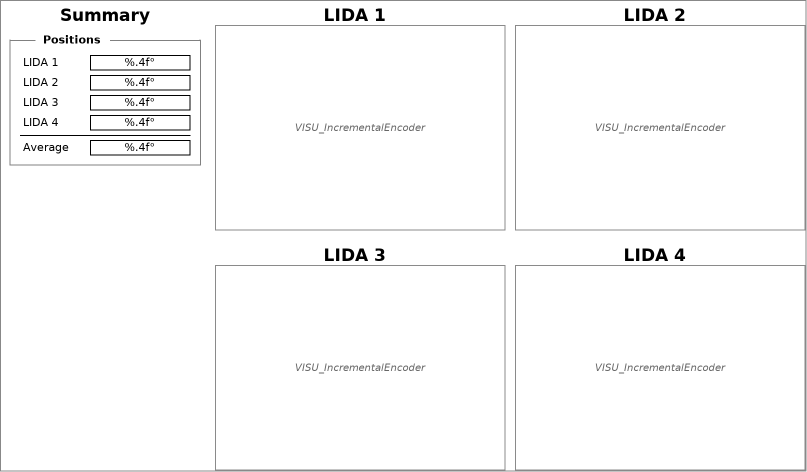
VISUALIZATION VISU_AxesAzimuthAxis_Lidas  // 807x472
VAR_IN_OUT
	ref : AxesAzimuthAxis;
    widget : AxesAzimuthAxisWidget;
END_VAR
    Label (215,0 280x30), "LIDA 1"
    Frame (215,25 290x205)
        shows VISU_IncrementalEncoder(ref := ref.parts.lida1, widget := widget.lida1)
    Label (215,240 280x30), "LIDA 3"
    Frame (215,265 290x205)
        shows VISU_IncrementalEncoder(ref := ref.parts.lida3, widget := widget.lida3)
    Label (515,0 280x30), "LIDA 2"
    Frame (515,25 290x205)
        shows VISU_IncrementalEncoder(ref := ref.parts.lida2, widget := widget.lida2)
    Label (515,240 280x30), "LIDA 4"
    Frame (515,265 290x205)
        shows VISU_IncrementalEncoder(ref := ref.parts.lida4, widget := widget.lida4)
    Label (10,0 190x30), "Summary"
    Label (40,30 65x20), "Positions"
    Polyline (110,40) (200,40) (200,165) (10,165) (10,40) (35,40)
    Label (20,55 90x15), "LIDA 1"
    Rectangle (90,55 100x15), "%.4f°", text variable: ref.lida1Position.degrees.value
    Rectangle (90,75 100x15), "%.4f°", text variable: ref.lida2Position.degrees.value
    Label (20,75 90x15), "LIDA 2"
    Rectangle (90,95 100x15), "%.4f°", text variable: ref.lida3Position.degrees.value
    Label (20,95 90x15), "LIDA 3"
    Rectangle (90,115 100x15), "%.4f°", text variable: ref.lida4Position.degrees.value
    Label (20,115 90x15), "LIDA 4"
    Label (20,140 90x15), "Average"
    Rectangle (90,140 100x15), "%.4f°", text variable: ref.lidaAveragePosition.degrees.value
    Line (20,135) (190,135)
END_VISUALIZATION

(* stored: Version 1.1.0.1, ProductVersion 3.1.4019.2
   Visu VISU_AxesAzimuthAxis_Lidas: Id {9438db80-1171-4a2e-880e-822a08e4787e} *)
